(* PLC project CoDeSys Library Template Interfaces, CODESYS CODESYS V3.5 SP16 Patch 1, author 3S - Smart Software Solutions GmbH *)
(* stored: creationDateTime 2022-10-04T11:36:41.0728712, version 3.5.16.0, modificationDateTime 2022-06-29T07:24:40.0702945, organization 3S - Smart Software Solutions GmbH *)
(* A interface library project template with all possible element types, docu and a sample project structure *)

{attribute 'qualified_only'}
{attribute 'strict'}
TYPE AXIS_DIRECTION : (DirectionPositive := 0, DirectionNegative := 1);
END_TYPE

{attribute 'qualified_only'}
{attribute 'strict'}
TYPE AXIS_STATUS : (ErrorStop := 0, Disabled := 1, Stopping := 2, Homing := 3, Standstill := 4, DiscreteMotion := 5, ContinuousMotion := 6, SynchronizedMotion := 7);
END_TYPE

{attribute 'qualified_only'}
{attribute 'strict'}
TYPE MC_BUFFER_MODE : (mcAborting := 0, mcBuffered := 1, mcBlendingLow := 2, mcBlendingPrevious := 3, mcBlendingNext := 4, mcBlendingHigh := 5);
END_TYPE

{attribute 'qualified_only'}
{attribute 'strict'}
TYPE MC_COMBINE_MODE : (enum_member := 0);
END_TYPE

{attribute 'qualified_only'}
{attribute 'strict'}
TYPE MC_Direction : (mcPositiveDirection := 0, mcShortestWay := 1, mcNegativeDirection := 2, mcCurrentDirection := 3);
END_TYPE

(* {attribute 'conditionalshow' := 'SomeText'} {attribute 'conditionalshow'} {attribute 'hide'} *)
{attribute 'qualified_only'}
TYPE MC_Error : (NO_ERROR, TIME_OUT);
END_TYPE

{attribute 'qualified_only'}
{attribute 'strict'}
TYPE MC_ExecutionMode : (mcImmediatly := 0, mcQueue := 1);
END_TYPE

{attribute 'qualified_only'}
{attribute 'strict'}
TYPE MC_Source : (mcSetValue := 0, mcActualValue := 1);
END_TYPE

{attribute 'qualified_only'}
{attribute 'strict'}
TYPE MC_StartMode : (mcAbsolute := 0, mcRelative := 1, mcRampIn := 2);
END_TYPE

{attribute 'qualified_only'}
{attribute 'strict'}
TYPE MC_SYNC_MODE : (enum_member := 0);
END_TYPE

{attribute 'qualified_only'}
{attribute 'strict'}
TYPE MOTION_STATUS : (ConstantVelocity := 0, Accelerating := 1, Decelerating := 2);
END_TYPE

TYPE MC_CAM_REF : STRUCT

END_STRUCT;
END_TYPE

TYPE MC_COMMAND_REF : STRUCT
  CommandId : INT;
END_STRUCT;
END_TYPE


INTERFACE itfAxis
METHOD Halt : itfAxisCommand
  VAR_INPUT
    Deceleration : REAL;
    Jerk : REAL;
    BufferMode : MC_BUFFER_MODE;
  END_VAR
END_METHOD
METHOD Home : itfAxisCommand
  VAR_INPUT
    Position : REAL;
    Velocity : REAL;
    EndVelocity : REAL;
    Acceleration : REAL;
    Deceleration : REAL;
    Jerk : REAL;
    Direction : MC_Direction;
    HomingMode : INT;
    BufferMode : MC_BUFFER_MODE;
  END_VAR
END_METHOD
METHOD MoveAbsolute : itfAxisCommand
  VAR_INPUT
    Position : REAL;
    Velocity : REAL;
    Acceleration : REAL;
    Deceleration : REAL;
    Jerk : REAL;
    Direction : MC_Direction;
    BufferMode : MC_BUFFER_MODE;
  END_VAR
END_METHOD
METHOD MoveSuperimposed : itfAxisCommand
  VAR_INPUT
    Distance : REAL;
    VelocityDiff : REAL;
    Acceleration : REAL;
    Deceleration : REAL;
    Jerk : REAL;
  END_VAR
END_METHOD
METHOD MoveRelative : itfAxisCommand
  VAR_INPUT
    Distance : REAL;
    Velocity : REAL;
    Acceleration : REAL;
    Deceleration : REAL;
    Jerk : REAL;
    BufferMode : MC_BUFFER_MODE;
  END_VAR
END_METHOD
METHOD MoveAdditive : itfAxisCommand
  VAR_INPUT
    Distance : REAL;
    Velocity : REAL;
    Acceleration : REAL;
    Deceleration : REAL;
    Jerk : REAL;
    BufferMode : MC_BUFFER_MODE;
  END_VAR
END_METHOD
METHOD MoveVelocity : itfContinuousAxisCommand
  VAR_INPUT
    Velocity : REAL;
    Acceleration : REAL;
    Deceleration : REAL;
    Jerk : REAL;
    Direction : MC_Direction;
    BufferMode : MC_BUFFER_MODE;
  END_VAR
END_METHOD
METHOD Stop : itfAxisCommand
  VAR_INPUT
    Deceleration : REAL;
    Jerk : REAL;
  END_VAR
END_METHOD
METHOD Reset : itfCommand
END_METHOD
METHOD Power : itfCommand
  VAR_INPUT
    Enable : BOOL;
    EnablePositive : BOOL;
    EnableNegative : BOOL;
  END_VAR
END_METHOD
METHOD ReadParameter : MC_Error
  VAR_INPUT
    ParameterNumber : INT;
  END_VAR
  VAR_OUTPUT
    Value : REAL;
  END_VAR
END_METHOD
METHOD ReadBoolParameter : MC_Error
  VAR_INPUT
    ParameterNumber : INT;
  END_VAR
  VAR_OUTPUT
    Value : BOOL;
  END_VAR
END_METHOD
METHOD WriteParameter : MC_Error
  VAR_INPUT
    ParameterNumber : INT;
    Value : REAL;
  END_VAR
END_METHOD
METHOD WriteBoolParameter : MC_Error
  VAR_INPUT
    ParameterNumber : INT;
    Value : BOOL;
  END_VAR
END_METHOD
METHOD SetPosition : itfCommand
  VAR_INPUT
    Position : REAL;
    Relative : BOOL;
    ExecutionMode : MC_ExecutionMode;
  END_VAR
END_METHOD
METHOD SetOverride : MC_Error
  VAR_INPUT
    VelFactor : REAL;
    AccFactor : REAL;
    JerkFactor : REAL;
  END_VAR
END_METHOD
METHOD GearIn : itfSynchronizedAxisCommand
  VAR_INPUT
    Master : itfAxis;
    Ratio : REAL;
    MasterValueSource : INT;
    Acceleration : REAL;
    Deceleration : REAL;
    Jerk : REAL;
    BufferMode : MC_BUFFER_MODE;
  END_VAR
END_METHOD
METHOD Release : MC_Error
END_METHOD
METHOD CamIn : itfSynchronizedAxisCommand
  VAR_INPUT
    Master : itfAxis;
    MasterOffset : REAL;
    SlaveOffset : REAL;
    MasterScaling : REAL;
    SlaveScaling : REAL;
    MasterStartDistance : REAL;
    MasterSyncPosition : REAL;
    StartMode : MC_StartMode;
    MasterValueSource : MC_Source;
    CamTable : itfCamTable;
    BufferMode : MC_BUFFER_MODE;
  END_VAR
END_METHOD
METHOD HaltSuperimposed : itfAxisCommand
  VAR_INPUT
    Deceleration : REAL;
    Jerk : REAL;
  END_VAR
END_METHOD
METHOD MoveContinuousAbsolute : itfContinuousAxisCommand
  VAR_INPUT
    Position : REAL;
    EndVelocity : REAL;
    Velocity : REAL;
    Acceleration : REAL;
    Deceleration : REAL;
    Jerk : REAL;
    Direction : MC_DIRECTION;
    BufferMode : MC_BUFFER_MODE;
  END_VAR
END_METHOD
METHOD MoveContinuousRelative : itfContinuousAxisCommand
  VAR_INPUT
    Distance : REAL;
    EndVelocity : REAL;
    Velocity : REAL;
    Acceleration : REAL;
    Deceleration : REAL;
    Jerk : REAL;
    Direction : MC_DIRECTION;
    BufferMode : MC_BUFFER_MODE;
  END_VAR
END_METHOD
METHOD TorqueControl : itfAxisCommand
  VAR_INPUT
    Torque : REAL;
    TorqueRamp : REAL;
    Velocity : REAL;
    Acceleration : REAL;
    Deceleration : REAL;
    Jerk : REAL;
    Direction : MC_DIRECTION;
    BufferMode : MC_BUFFER_MODE;
  END_VAR
END_METHOD
METHOD PositionProfile : itfCommand
  VAR_INPUT
    TimeScale : REAL;
    PositionScale : REAL;
    Offset : REAL;
    BufferMode : MC_BUFFER_MODE;
  END_VAR
END_METHOD
METHOD VelocityProfile : itfCommand
  VAR_INPUT
    TimeScale : REAL;
    VelocityScale : REAL;
    Offset : REAL;
    BufferMode : MC_BUFFER_MODE;
  END_VAR
END_METHOD
METHOD AccelerationProfile : itfCommand
  VAR_INPUT
    TimeScale : REAL;
    AccelerationScale : REAL;
    Offset : REAL;
    BufferMode : MC_BUFFER_MODE;
  END_VAR
END_METHOD
METHOD GearInPos : itfSynchronizedAxisCommand
  VAR_INPUT
    Master : itfAxis;
    RatioNumerator : REAL;
    RatioDenominator : REAL;
    MasterValueSource : MC_SOURCE;
    MasterSyncPosition : REAL;
    SlaveSyncPosition : REAL;
    SyncMode : MC_SYNC_MODE;
    MasterStartDistance : REAL;
    Velocity : REAL;
    Acceleration : REAL;
    Deceleration : REAL;
    Jerk : REAL;
    BufferMode : MC_BUFFER_MODE;
  END_VAR
END_METHOD
METHOD PhasingAbsolute : itfSynchronizedAxisCommand
  VAR_INPUT
    Master : itfAxis;
    PhaseShift : REAL;
    Velocity : REAL;
    Acceleration : REAL;
    Deceleration : REAL;
    Jerk : REAL;
    BufferMode : MC_BUFFER_MODE;
  END_VAR
END_METHOD
METHOD PhasingRelative : itfSynchronizedAxisCommand
  VAR_INPUT
    Master : itfAxis;
    PhaseShift : REAL;
    Velocity : REAL;
    Acceleration : REAL;
    Deceleration : REAL;
    Jerk : REAL;
    BufferMode : MC_BUFFER_MODE;
  END_VAR
END_METHOD
METHOD CombineAxes : itfSynchronizedAxisCommand
  VAR_INPUT
    Master1 : itfAxis;
    Master2 : itfAxis;
    CombineMode : MC_COMBINE_MODE;
    GearRatioNumeratorM1 : INT;
    GearRatioDenominatorM1 : INT;
    GearRatioNumeratorM2 : INT;
    GearRatioDenominatorM2 : INT;
    MasterValueSourceM1 : MC_SOURCE;
    MasterValueSourceM2 : MC_SOURCE;
    BufferMode : MC_BUFFER_MODE;
  END_VAR
END_METHOD
PROPERTY HomeAbsSwitch : BOOL
END_PROPERTY
PROPERTY LimitSwitchPositive : BOOL
END_PROPERTY
PROPERTY LimitSwitchNegative : BOOL
END_PROPERTY
PROPERTY Simulation : BOOL
END_PROPERTY
PROPERTY CommunicationReady : BOOL
END_PROPERTY
PROPERTY ReadyForPowerOn : BOOL
END_PROPERTY
PROPERTY PowerOn : BOOL
END_PROPERTY
PROPERTY IsHomed : BOOL
END_PROPERTY
PROPERTY AxisWarning : BOOL
END_PROPERTY
PROPERTY ErrorId : WORD
END_PROPERTY
PROPERTY Status : AXIS_STATUS
END_PROPERTY
PROPERTY MotionStatus : MOTION_STATUS
END_PROPERTY
PROPERTY Direction : AXIS_DIRECTION
END_PROPERTY
PROPERTY ActualPosition : REAL
END_PROPERTY
PROPERTY ActualVelocity : REAL
END_PROPERTY
PROPERTY ActualTorque : REAL
END_PROPERTY
END_INTERFACE

INTERFACE itfAxisCommand
METHOD Update : MC_Error
  VAR_INPUT
    Position : REAL;
    Velocity : REAL;
    EndVelocity : REAL;
    Acceleration : REAL;
    Deceleration : REAL;
    Jerk : REAL;
  END_VAR
END_METHOD
END_INTERFACE

INTERFACE itfCamTable
METHOD Select : itfCommand
  VAR_INPUT
    Periodic : BOOL;
    MasterAbsolute : BOOL;
    SlaveAbsolute : BOOL;
    CamTable : MC_CAM_REF;
  END_VAR
END_METHOD
END_INTERFACE

INTERFACE itfCommand
METHOD Abort : MC_Error
END_METHOD
METHOD Wait : MC_Error
  VAR_INPUT
    Timeout : TIME;
    AbortOnTimeout : BOOL;
  END_VAR
END_METHOD
PROPERTY Command : MC_COMMAND_REF
END_PROPERTY
PROPERTY Done : BOOL
END_PROPERTY
PROPERTY Busy : BOOL
END_PROPERTY
PROPERTY Active : BOOL
END_PROPERTY
PROPERTY CommandAborted : BOOL
END_PROPERTY
PROPERTY Error : BOOL
END_PROPERTY
PROPERTY ErrorId : MC_Error
END_PROPERTY
END_INTERFACE

INTERFACE itfContinuousAxisCommand
PROPERTY InVelocity : BOOL
END_PROPERTY
END_INTERFACE

INTERFACE itfSynchronizedAxisCommand
PROPERTY InSync : BOOL
END_PROPERTY
END_INTERFACE

PROGRAM CamGearExample
  VAR
    MasterDrive : Axis;  (* Hardware definitions *)
    CamDrive : Axis;
    GearDrive : Axis;
    Table : CamTable;
    TableData : MC_CAM_REF;
    Velocity : REAL := 5;
    MasterState : INT := 0;  (* States *)
    CamState : INT := 0;
    GearState : INT := 0;
    Start : BOOL := FALSE;  (* Control *)
    MasterMove : itfCommand;  (* Commands *)
    TableSet : itfCommand;
    CamMove : itfSynchronizedAxisCommand;
    GearMove : itfSynchronizedAxisCommand;
  END_VAR

            CASE MasterState OF
	0: // Disabled
		IF Start THEN
			MasterState := MasterState + 1;
		END_IF
		
	1: // Power On
		MasterDrive.Power(Enable:=TRUE, EnablePositive:=TRUE, EnableNegative:=TRUE);
		IF MasterDrive.Status = AXIS_STATUS.Standstill THEN
			MasterState := MasterState + 1;
		END_IF
		
	2: // Wait for other drives 
		IF CamMove.InSync AND GearMove.InSync THEN
			MasterMove := MasterDrive.MoveVelocity(Velocity:=Velocity, Acceleration:=0, Deceleration:=0, Jerk:=0, Direction:=MC_Direction.mcPositiveDirection, BufferMode:=MC_BUFFER_MODE.mcAborting);
			MasterState := MasterState + 1;
		END_IF
		
	3: // Moving
		IF NOT Start THEN
			MasterMove:= MasterDrive.Halt(Deceleration:=0, Jerk:=0, BufferMode:=MC_BUFFER_MODE.mcAborting);
			MasterState := MasterState + 1;
		END_IF
		
	4: // Stopping
		IF NOT MasterMove.Done THEN
			MasterState := MasterState + 1;
		END_IF
		
	5: // Power off
		MasterDrive.Power(Enable:=FALSE, EnablePositive:=FALSE, EnableNegative:=FALSE);
		IF MasterDrive.Status = AXIS_STATUS.Disabled THEN
			MasterState := 0;
		END_IF
END_CASE

CASE CamState OF
	0: // Disabled
		IF Start THEN
			CamState := CamState + 1;
		END_IF
		
	1: // Power On
		CamDrive.Power(Enable:=TRUE, EnablePositive:=TRUE, EnableNegative:=TRUE);
		IF CamDrive.Status = AXIS_STATUS.Standstill AND MasterDrive.Status = AXIS_STATUS.Standstill THEN
			TableSet := Table.Select(CamTable:=TableData, Periodic:=TRUE, MasterAbsolute:=TRUE, SlaveAbsolute:=TRUE);
			CamState := CamState + 1;
		END_IF
		
	2: // Set CAM Table
		IF TableSet.Done THEN
			CamMove := CamDrive.CamIn(Master:=MasterDrive, MasterOffset:=0, SlaveOffset:=0, MasterScaling:=1, SlaveScaling:=1, MasterStartDistance:=0, MasterSyncPosition:=0, 
				StartMode:=MC_StartMode.mcRelative, MasterValueSource:=MC_Source.mcSetValue,CamTable:=Table, BufferMode:=MC_BUFFER_MODE.mcAborting);
			CamState := CamState + 1;
		END_IF
		
	3: // Synchronized
		IF NOT Start THEN
			CamDrive.Release();
			CamState := CamState + 1;
		END_IF
		
	4: // Power off
		CamDrive.Power(Enable:=FALSE, EnablePositive:=FALSE, EnableNegative:=FALSE);
		IF CamDrive.Status = AXIS_STATUS.Disabled THEN
			CamState := 0;
		END_IF
END_CASE

CASE GearState OF
	0: // Disabled
		IF Start THEN
			GearState := GearState + 1;
		END_IF
		
	1: // Power On
		GearDrive.Power(Enable:=TRUE, EnablePositive:=TRUE, EnableNegative:=TRUE);
		IF GearDrive.Status = AXIS_STATUS.Standstill AND MasterDrive.Status = AXIS_STATUS.Standstill THEN
			GearMove := GearDrive.GearIn(Master:=MasterDrive, Ratio:=2, MasterValueSource:=MC_Source.mcSetValue,Acceleration:=0, Deceleration:=0, Jerk:=0, BufferMode:=MC_BUFFER_MODE.mcAborting);
			GearState := GearState + 1;
		END_IF
		
	2: // Synchronized
		IF NOT Start THEN
			GearDrive.Release();
			GearState := GearState + 1;
		END_IF
		
	3: // Power off
		GearDrive.Power(Enable:=FALSE, EnablePositive:=FALSE, EnableNegative:=FALSE);
		IF GearDrive.Status = AXIS_STATUS.Disabled THEN
			GearState := 0;
		END_IF
END_CASE

          
END_PROGRAM

PROGRAM LabelingExample
  VAR
    LabelDrive : Axis;  (* Hardware definitions *)
    Conveyor : Axis;
    LabelLength : REAL := 100;
    SensorDistance : REAL := 10;
    Velocity : REAL := 5;
    ProductDetection : BOOL := FALSE;
    DelayTimer : TON;
    ConveyorState : INT := 0;  (* States *)
    LabelDriveState : INT := 0;
    Start : BOOL := FALSE;  (* Control *)
    ConveyorMove : itfCommand;  (* Commands *)
    LabelDriveMove : itfCommand;
  END_VAR

            // Run the timer. As it is a classic FB it should be called every cycle
DelayTimer(IN:=ProductDetection, PT:= INT_TO_TIME(REAL_TO_INT(SensorDistance * 1000 / Velocity)));

CASE ConveyorState OF
	0: // Disabled
		IF Start THEN
			ConveyorState := ConveyorState + 1;
		END_IF
		
	1: // Power On
		Conveyor.Power(Enable:=TRUE, EnablePositive:=TRUE, EnableNegative:=TRUE);
		IF Conveyor.Status = AXIS_STATUS.Standstill THEN
			ConveyorState := ConveyorState + 1;
		END_IF
		
	2: // Wait for LabelDrive 
		IF LabelDrive.Status = AXIS_STATUS.Standstill THEN
			ConveyorMove := Conveyor.MoveVelocity(Velocity:=Velocity, Acceleration:=0, Deceleration:=0, Jerk:=0, Direction:=MC_Direction.mcPositiveDirection, BufferMode:=MC_BUFFER_MODE.mcAborting);
			ConveyorState := ConveyorState + 1;
		END_IF
		
	3: // Moving
		IF NOT Start THEN
			ConveyorMove := Conveyor.Halt(Deceleration:=0, Jerk:=0, BufferMode:=MC_BUFFER_MODE.mcAborting);
			ConveyorState := ConveyorState + 1;
		END_IF
		
	4: // Stopping
		IF ConveyorMove.Done THEN
			ConveyorState := ConveyorState + 1;
		END_IF
		
	5: // Power off
		Conveyor.Power(Enable:=FALSE, EnablePositive:=FALSE, EnableNegative:=FALSE);
		IF Conveyor.Status = AXIS_STATUS.Disabled THEN
			ConveyorState := 0;
		END_IF
END_CASE

CASE LabelDriveState OF
	0: // Disabled
		IF Start THEN
			LabelDriveState := LabelDriveState + 1;
		END_IF
		
	1: // Power On
		LabelDrive.Power(Enable:=TRUE, EnablePositive:=TRUE, EnableNegative:=TRUE);
		IF LabelDrive.Status = AXIS_STATUS.Standstill THEN
			LabelDriveState := LabelDriveState + 1;
		END_IF
		
	2: // Wait for Conveyor 
		IF Conveyor.Status = AXIS_STATUS.Standstill THEN
			LabelDriveState := LabelDriveState + 1;
		END_IF
		
	3: // Wait for product
		IF NOT Start THEN
			LabelDriveState := 5;
		END_IF
		IF DelayTimer.Q THEN
			LabelDriveMove := LabelDrive.MoveRelative(Distance:=LabelLength, Velocity:=Velocity, Acceleration:=0, Deceleration:=0, Jerk:=0, BufferMode:=MC_BUFFER_MODE.mcAborting);
			LabelDriveState := LabelDriveState + 1;
		END_IF
		
	4: // Wait for label to be transfered
		IF LabelDriveMove.Done AND NOT DelayTimer.Q THEN
			LabelDriveState := 3;
		END_IF
		
	5: // Power off
		Conveyor.Power(Enable:=FALSE, EnablePositive:=FALSE, EnableNegative:=FALSE);
		IF Conveyor.Status = AXIS_STATUS.Disabled THEN
			LabelDriveState := 0;
		END_IF
	
END_CASE

          
END_PROGRAM

PROGRAM WarehousingExample
  VAR
    Axis_X : itfAxis;
    Axis_Y : itfAxis;
    Axis_Z : itfAxis;
    stateOOP : INT;
    lastCommandX : itfCommand;
    lastCommandY : itfCommand;
    lastCommandZ : itfCommand;
    stepOn : BOOL := FALSE;
    targetPosX : REAL := 400;
    targetPosY : REAL := 600;
  END_VAR

            CASE stateOOP OF
	0: ;
	10: 
	// init
		Axis_X.Power(Enable:=TRUE, EnablePositive:=TRUE, EnableNegative:=TRUE);
		Axis_Y.Power(Enable:=TRUE, EnablePositive:=TRUE, EnableNegative:=TRUE);
		Axis_Z.Power(Enable:=TRUE, EnablePositive:=TRUE, EnableNegative:=TRUE);
	
		IF stepOn THEN
			stateOOP := stateOOP + 10;
		END_IF
	20:
	// start movement in XY
		lastCommandX := Axis_X.MoveAbsolute(Position:=targetPosX, Velocity:=40, Acceleration:=0, Deceleration:=0, Jerk:=0, Direction:=0, BufferMode:=MC_BUFFER_MODE.mcAborting);
		lastCommandY := Axis_Y.MoveAbsolute(Position:=targetPosY, Velocity:=40, Acceleration:=0, Deceleration:=0, Jerk:=0, Direction:=0, BufferMode:=MC_BUFFER_MODE.mcAborting);
		stateOOP := stateOOP + 10;
	30:
	// wait till movement is finished to 'forkIn'
		IF lastCommandX.Done AND lastCommandY.Done THEN
			lastCommandZ := Axis_Z.MoveRelative(Distance:=100, Velocity:=20, Acceleration:=0, Deceleration:=0, Jerk:=0, BufferMode:=MC_BUFFER_MODE.mcAborting);
			stateOOP := stateOOP + 10;
		END_IF
	40:
	// lift pallet if forked in
		IF lastCommandZ.Done THEN
			lastCommandY := Axis_Y.MoveRelative(Distance:=100, Velocity:=10, Acceleration:=0, Deceleration:=0, Jerk:=0, BufferMode:=MC_BUFFER_MODE.mcAborting);
			stateOOP := stateOOP + 10;
		END_IF
	50:
	// fork out with pallet if forked in is done
		IF lastCommandY.Done THEN
			lastCommandZ := Axis_Z.MoveAbsolute(Position:=0, Velocity:=20, Acceleration:=0, Deceleration:=0, Jerk:=0, Direction:=0, BufferMode:=MC_BUFFER_MODE.mcAborting);
			stateOOP := stateOOP + 10;
		END_IF
	60:
	// move to delivery if fork out is done
		IF lastCommandZ.Done THEN
			lastCommandX := Axis_X.MoveAbsolute(Position:=0, Velocity:=40, Acceleration:=0, Deceleration:=0, Jerk:=0, Direction:=0, BufferMode:=MC_BUFFER_MODE.mcAborting);
			lastCommandY := Axis_Y.MoveAbsolute(Position:=0, Velocity:=40, Acceleration:=0, Deceleration:=0, Jerk:=0, Direction:=0, BufferMode:=MC_BUFFER_MODE.mcAborting);
			stateOOP := stateOOP + 10;
		END_IF
	70:
	// wait till finished
		IF lastCommandX.Done AND lastCommandY.Done THEN
			stateOOP := stateOOP + 10;
		END_IF
	80: 
	// ready
	;
END_CASE
          
END_PROGRAM
